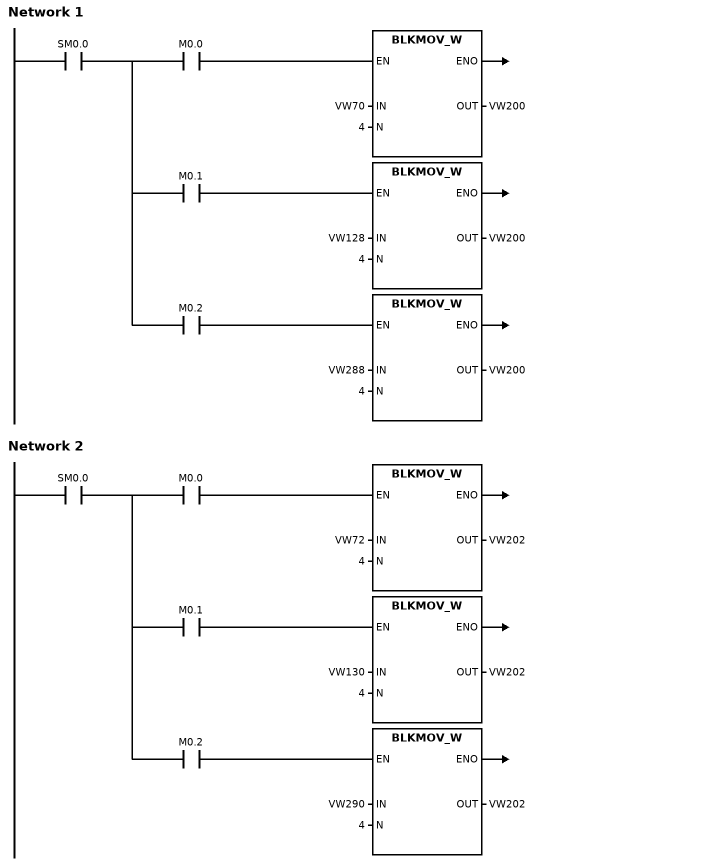
Network 1
LD     SM0.0
LPS
A      M0.0
BMW    VW70, VW200, 4
LRD
A      M0.1
BMW    VW128, VW200, 4
LPP
A      M0.2
BMW    VW288, VW200, 4
Network 2
LD     SM0.0
LPS
A      M0.0
BMW    VW72, VW202, 4
LRD
A      M0.1
BMW    VW130, VW202, 4
LPP
A      M0.2
BMW    VW290, VW202, 4
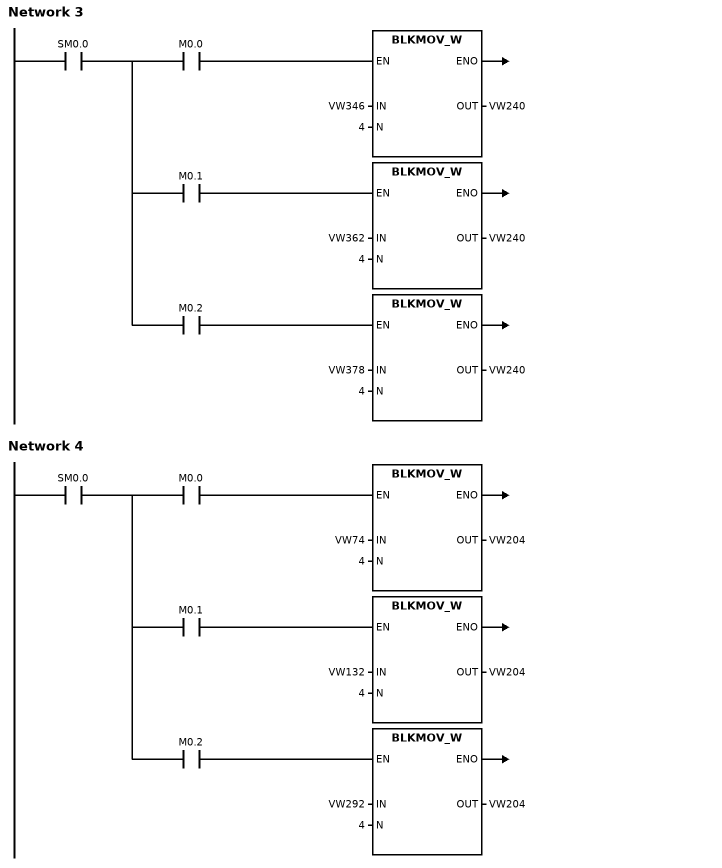
Network 3
LD     SM0.0
LPS
A      M0.0
BMW    VW346, VW240, 4
LRD
A      M0.1
BMW    VW362, VW240, 4
LPP
A      M0.2
BMW    VW378, VW240, 4
Network 4
LD     SM0.0
LPS
A      M0.0
BMW    VW74, VW204, 4
LRD
A      M0.1
BMW    VW132, VW204, 4
LPP
A      M0.2
BMW    VW292, VW204, 4
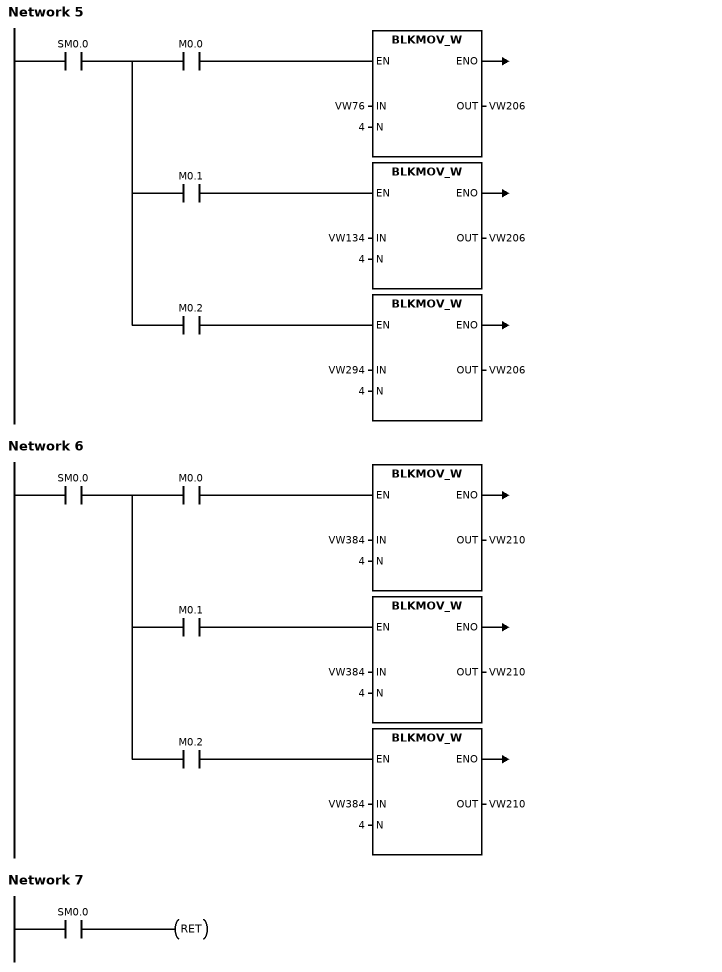
Network 5
LD     SM0.0
LPS
A      M0.0
BMW    VW76, VW206, 4
LRD
A      M0.1
BMW    VW134, VW206, 4
LPP
A      M0.2
BMW    VW294, VW206, 4
Network 6
LD     SM0.0
LPS
A      M0.0
BMW    VW384, VW210, 4
LRD
A      M0.1
BMW    VW384, VW210, 4
LPP
A      M0.2
BMW    VW384, VW210, 4
Network 7
LD     SM0.0
CRET
END_SUBROUTINE_BLOCK

SUBROUTINE_BLOCK thoidiem7:SBR9
TITLE=
BEGIN
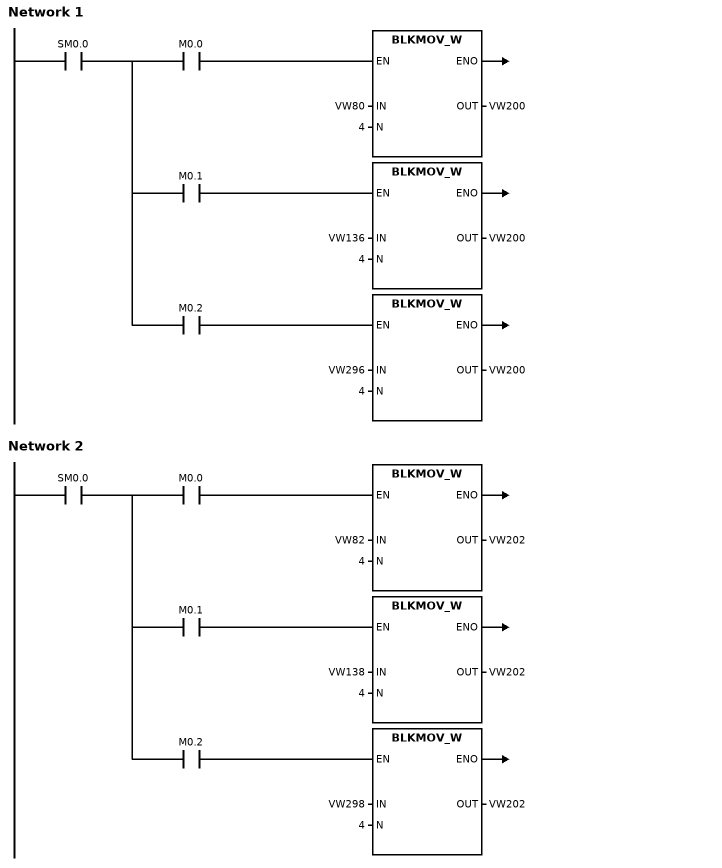
Network 1
LD     SM0.0
LPS
A      M0.0
BMW    VW80, VW200, 4
LRD
A      M0.1
BMW    VW136, VW200, 4
LPP
A      M0.2
BMW    VW296, VW200, 4
Network 2
LD     SM0.0
LPS
A      M0.0
BMW    VW82, VW202, 4
LRD
A      M0.1
BMW    VW138, VW202, 4
LPP
A      M0.2
BMW    VW298, VW202, 4
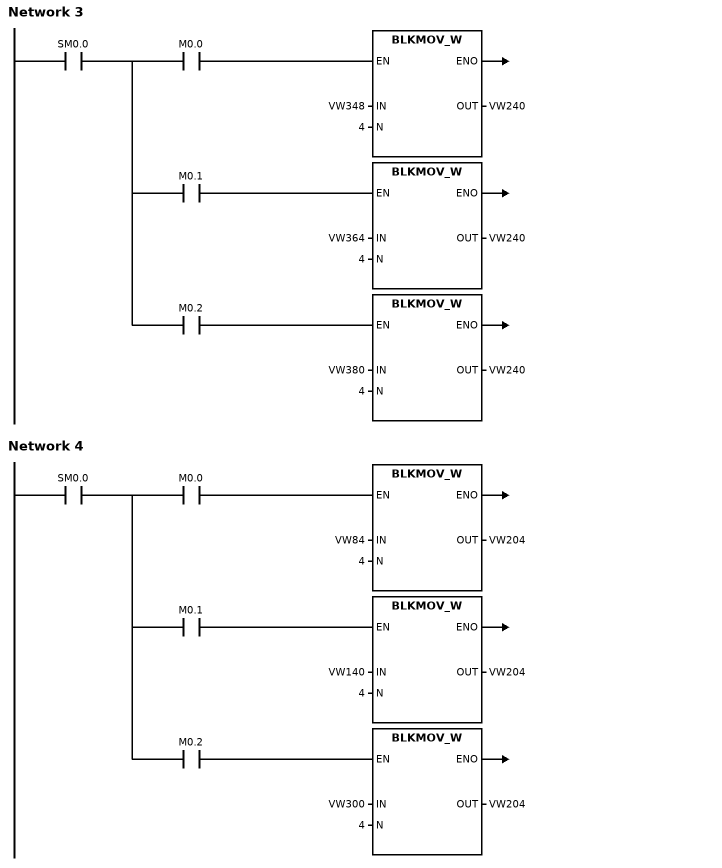
Network 3
LD     SM0.0
LPS
A      M0.0
BMW    VW348, VW240, 4
LRD
A      M0.1
BMW    VW364, VW240, 4
LPP
A      M0.2
BMW    VW380, VW240, 4
Network 4
LD     SM0.0
LPS
A      M0.0
BMW    VW84, VW204, 4
LRD
A      M0.1
BMW    VW140, VW204, 4
LPP
A      M0.2
BMW    VW300, VW204, 4
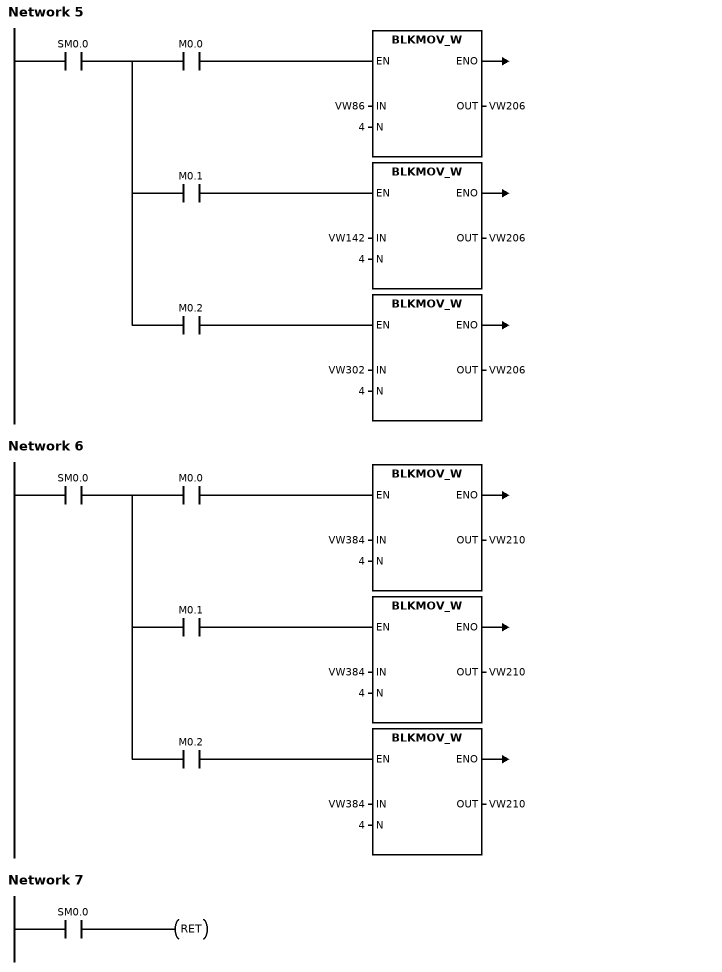
Network 5
LD     SM0.0
LPS
A      M0.0
BMW    VW86, VW206, 4
LRD
A      M0.1
BMW    VW142, VW206, 4
LPP
A      M0.2
BMW    VW302, VW206, 4
Network 6
LD     SM0.0
LPS
A      M0.0
BMW    VW384, VW210, 4
LRD
A      M0.1
BMW    VW384, VW210, 4
LPP
A      M0.2
BMW    VW384, VW210, 4
Network 7
LD     SM0.0
CRET
END_SUBROUTINE_BLOCK

SUBROUTINE_BLOCK tudong3phase:SBR10
TITLE=
BEGIN
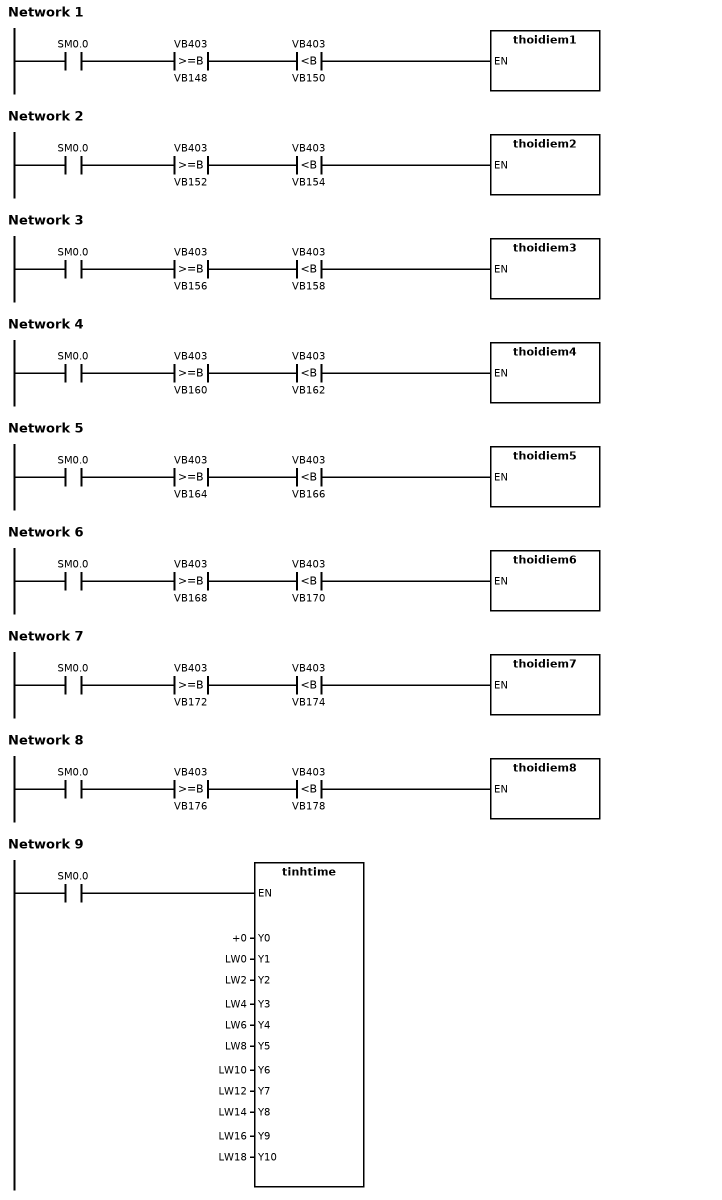
Network 1
LD     SM0.0
AB>=   VB403, VB148
AB<    VB403, VB150
CALL   thoidiem1:SBR3
Network 2
LD     SM0.0
AB>=   VB403, VB152
AB<    VB403, VB154
CALL   thoidiem2:SBR4
Network 3
LD     SM0.0
AB>=   VB403, VB156
AB<    VB403, VB158
CALL   thoidiem3:SBR5
Network 4
LD     SM0.0
AB>=   VB403, VB160
AB<    VB403, VB162
CALL   thoidiem4:SBR6
Network 5
LD     SM0.0
AB>=   VB403, VB164
AB<    VB403, VB166
CALL   thoidiem5:SBR7
Network 6
LD     SM0.0
AB>=   VB403, VB168
AB<    VB403, VB170
CALL   thoidiem6:SBR8
Network 7
LD     SM0.0
AB>=   VB403, VB172
AB<    VB403, VB174
CALL   thoidiem7:SBR9
Network 8
LD     SM0.0
AB>=   VB403, VB176
AB<    VB403, VB178
CALL   thoidiem8:SBR14
Network 9
LD     SM0.0
CALL   tinhtime:SBR16, +0, LW0, LW2, LW4, LW6, LW8, LW10, LW12, LW14, LW16, LW18
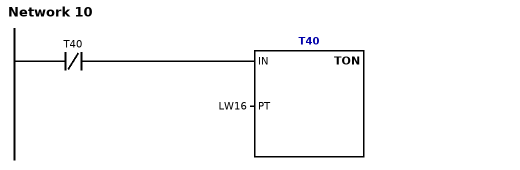
Network 10
LDN    T40
TON    T40, LW16
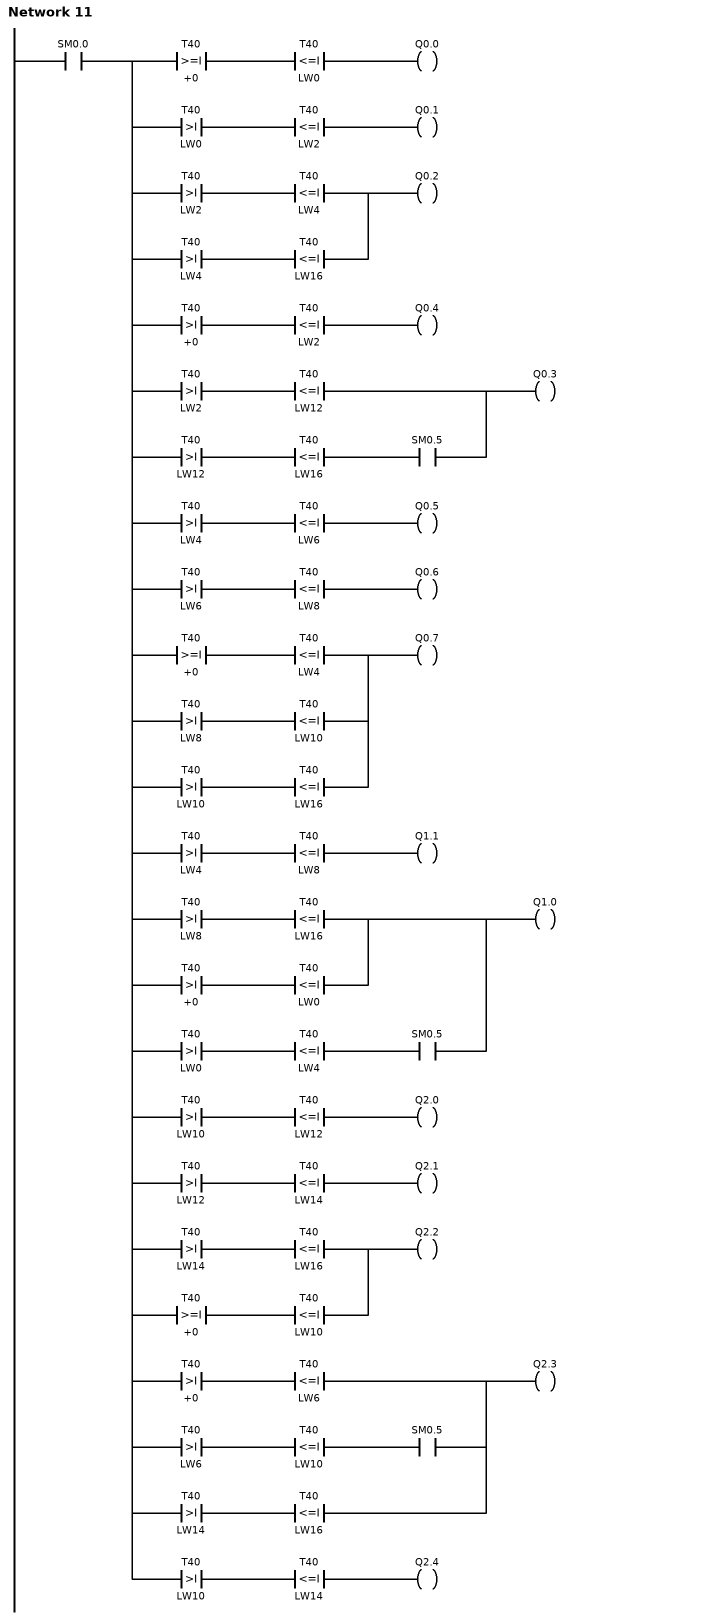
Network 11
LD     SM0.0
LPS
AW>=   T40, +0
AW<=   T40, LW0
=      Q0.0
LRD
AW>    T40, LW0
AW<=   T40, LW2
=      Q0.1
LRD
LDW>   T40, LW2
AW<=   T40, LW4
LDW>   T40, LW4
AW<=   T40, LW16
OLD
ALD
=      Q0.2
LRD
AW>    T40, +0
AW<=   T40, LW2
=      Q0.4
LRD
LDW>   T40, LW2
AW<=   T40, LW12
LDW>   T40, LW12
AW<=   T40, LW16
A      SM0.5
OLD
ALD
=      Q0.3
LRD
LPS
AW>    T40, LW4
AW<=   T40, LW6
=      Q0.5
LPP
AW>    T40, LW6
AW<=   T40, LW8
=      Q0.6
LRD
LDW>=  T40, +0
AW<=   T40, LW4
LDW>   T40, LW8
AW<=   T40, LW10
OLD
LDW>   T40, LW10
AW<=   T40, LW16
OLD
ALD
=      Q0.7
LRD
AW>    T40, LW4
AW<=   T40, LW8
=      Q1.1
LRD
LDW>   T40, LW8
AW<=   T40, LW16
LDW>   T40, +0
AW<=   T40, LW0
OLD
LDW>   T40, LW0
AW<=   T40, LW4
A      SM0.5
OLD
ALD
=      Q1.0
LRD
LPS
AW>    T40, LW10
AW<=   T40, LW12
=      Q2.0
LPP
AW>    T40, LW12
AW<=   T40, LW14
=      Q2.1
LRD
LDW>   T40, LW14
AW<=   T40, LW16
LDW>=  T40, +0
AW<=   T40, LW10
OLD
ALD
=      Q2.2
LRD
LDW>   T40, +0
AW<=   T40, LW6
LDW>   T40, LW6
AW<=   T40, LW10
A      SM0.5
OLD
LDW>   T40, LW14
AW<=   T40, LW16
OLD
ALD
=      Q2.3
LPP
AW>    T40, LW10
AW<=   T40, LW14
=      Q2.4
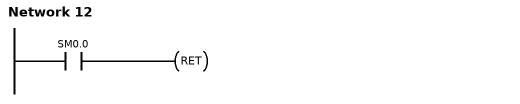
Network 12
LD     SM0.0
CRET
END_SUBROUTINE_BLOCK

SUBROUTINE_BLOCK chonngay:SBR11
TITLE=
BEGIN
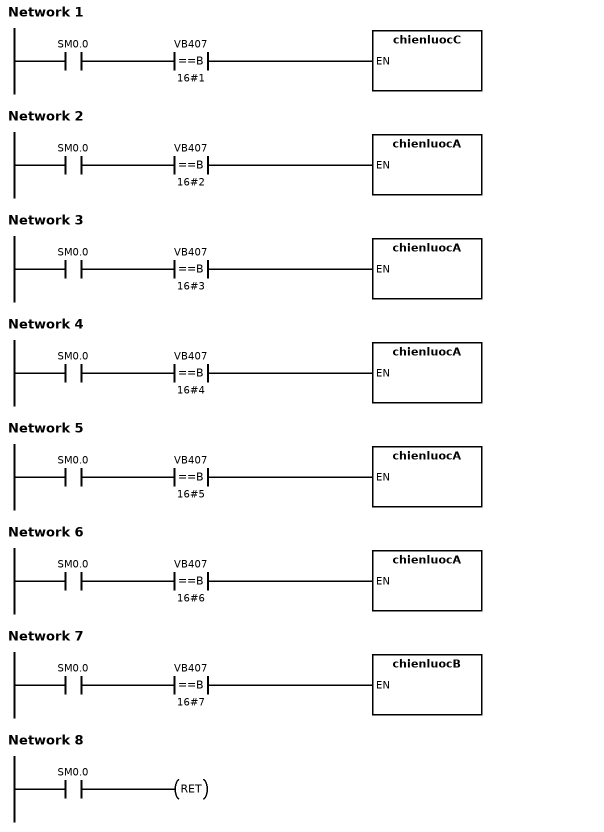
Network 1
LD     SM0.0
AB=    VB407, 16#1
CALL   chienluocC:SBR15
Network 2
LD     SM0.0
AB=    VB407, 16#2
CALL   chienluocA:SBR12
Network 3
LD     SM0.0
AB=    VB407, 16#3
CALL   chienluocA:SBR12
Network 4
LD     SM0.0
AB=    VB407, 16#4
CALL   chienluocA:SBR12
Network 5
LD     SM0.0
AB=    VB407, 16#5
CALL   chienluocA:SBR12
Network 6
LD     SM0.0
AB=    VB407, 16#6
CALL   chienluocA:SBR12
Network 7
LD     SM0.0
AB=    VB407, 16#7
CALL   chienluocB:SBR13
Network 8
LD     SM0.0
CRET
END_SUBROUTINE_BLOCK

SUBROUTINE_BLOCK chienluocA:SBR12
TITLE=
BEGIN
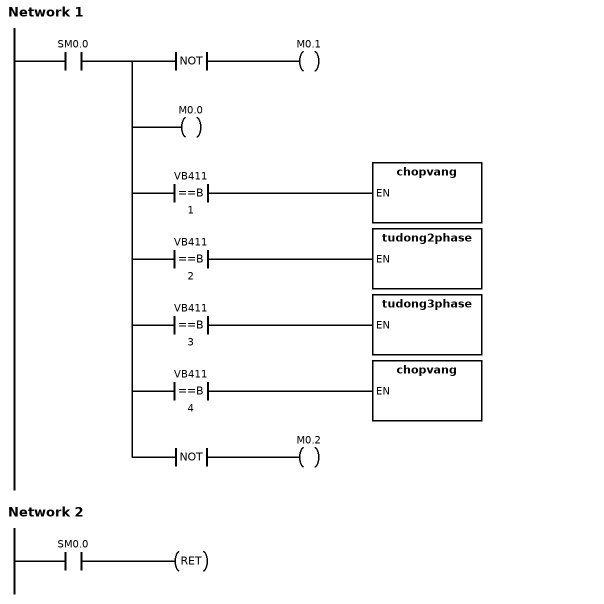
Network 1
LD     SM0.0
LPS
NOT
=      M0.1
LRD
=      M0.0
LRD
AB=    VB411, 1
CALL   chopvang:SBR1
LRD
AB=    VB411, 2
CALL   tudong2phase:SBR0
LRD
AB=    VB411, 3
CALL   tudong3phase:SBR10
LRD
AB=    VB411, 4
CALL   chopvang:SBR1
LPP
NOT
=      M0.2
Network 2
LD     SM0.0
CRET
END_SUBROUTINE_BLOCK

SUBROUTINE_BLOCK chienluocB:SBR13
TITLE=
BEGIN
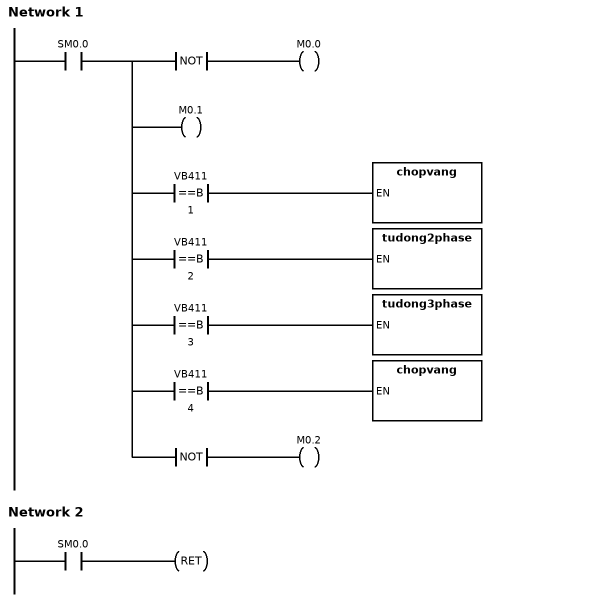
Network 1
LD     SM0.0
LPS
NOT
=      M0.0
LRD
=      M0.1
LRD
AB=    VB411, 1
CALL   chopvang:SBR1
LRD
AB=    VB411, 2
CALL   tudong2phase:SBR0
LRD
AB=    VB411, 3
CALL   tudong3phase:SBR10
LRD
AB=    VB411, 4
CALL   chopvang:SBR1
LPP
NOT
=      M0.2
Network 2
LD     SM0.0
CRET
END_SUBROUTINE_BLOCK

SUBROUTINE_BLOCK thoidiem8:SBR14
TITLE=
BEGIN
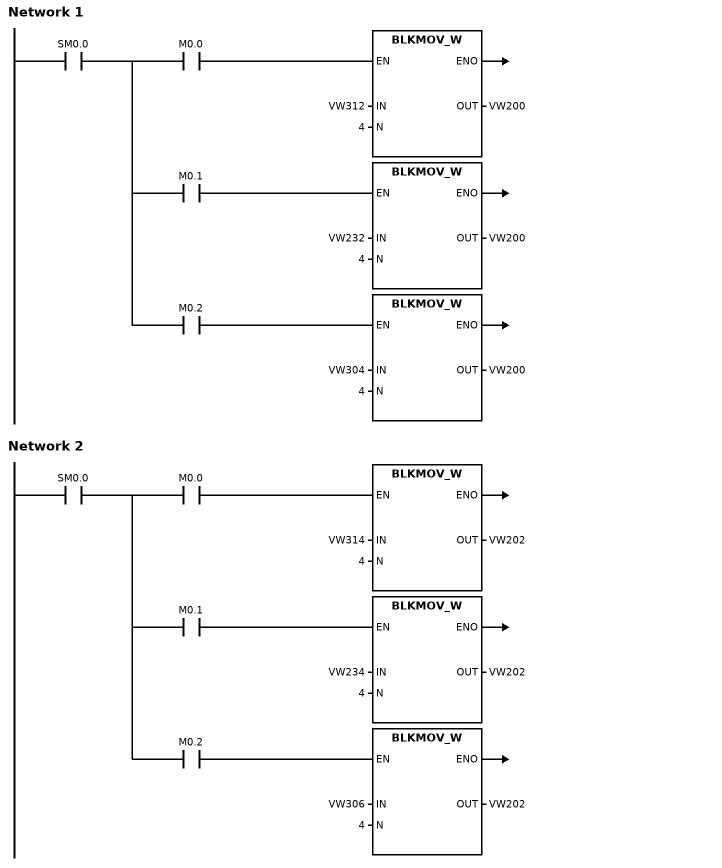
Network 1
LD     SM0.0
LPS
A      M0.0
BMW    VW312, VW200, 4
LRD
A      M0.1
BMW    VW232, VW200, 4
LPP
A      M0.2
BMW    VW304, VW200, 4
Network 2
LD     SM0.0
LPS
A      M0.0
BMW    VW314, VW202, 4
LRD
A      M0.1
BMW    VW234, VW202, 4
LPP
A      M0.2
BMW    VW306, VW202, 4
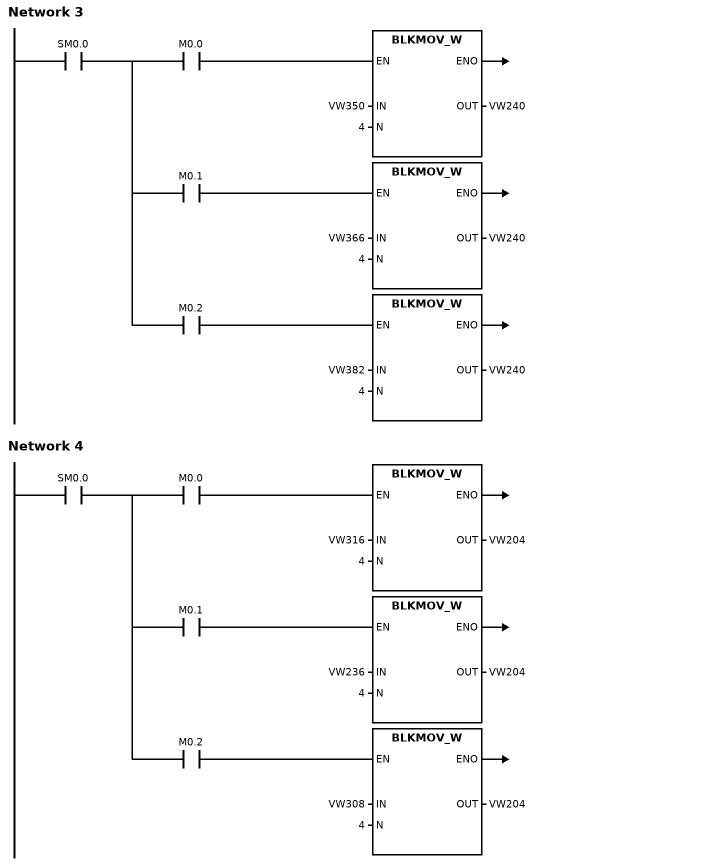
Network 3
LD     SM0.0
LPS
A      M0.0
BMW    VW350, VW240, 4
LRD
A      M0.1
BMW    VW366, VW240, 4
LPP
A      M0.2
BMW    VW382, VW240, 4
Network 4
LD     SM0.0
LPS
A      M0.0
BMW    VW316, VW204, 4
LRD
A      M0.1
BMW    VW236, VW204, 4
LPP
A      M0.2
BMW    VW308, VW204, 4
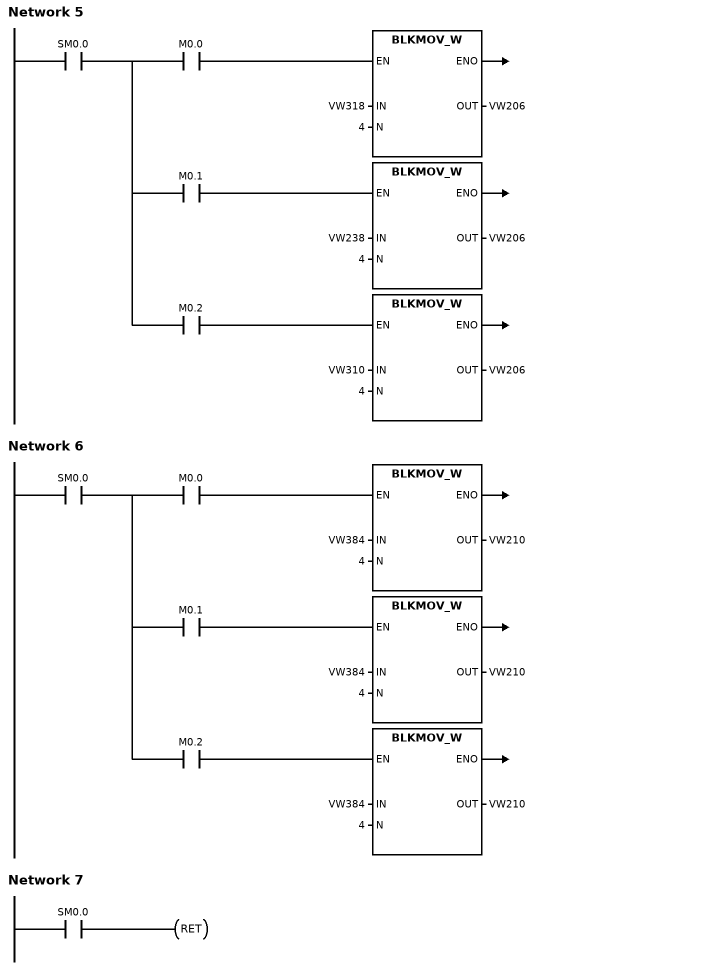
Network 5
LD     SM0.0
LPS
A      M0.0
BMW    VW318, VW206, 4
LRD
A      M0.1
BMW    VW238, VW206, 4
LPP
A      M0.2
BMW    VW310, VW206, 4
Network 6
LD     SM0.0
LPS
A      M0.0
BMW    VW384, VW210, 4
LRD
A      M0.1
BMW    VW384, VW210, 4
LPP
A      M0.2
BMW    VW384, VW210, 4
Network 7
LD     SM0.0
CRET
END_SUBROUTINE_BLOCK

SUBROUTINE_BLOCK chienluocC:SBR15
TITLE=
BEGIN
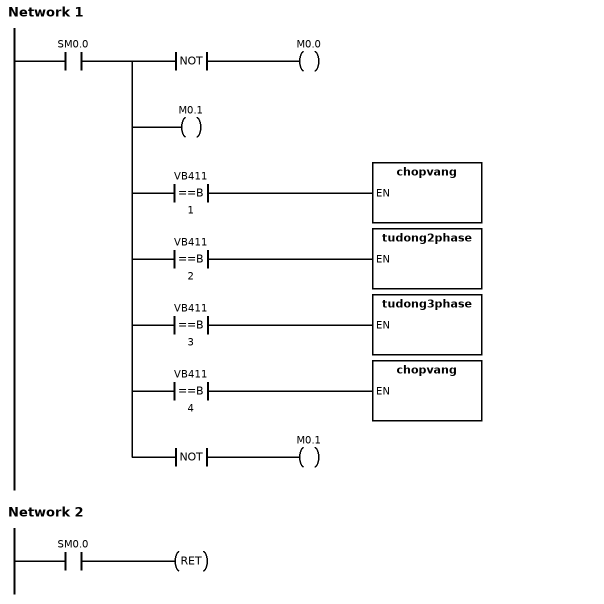
Network 1
LD     SM0.0
LPS
NOT
=      M0.0
LRD
=      M0.1
LRD
AB=    VB411, 1
CALL   chopvang:SBR1
LRD
AB=    VB411, 2
CALL   tudong2phase:SBR0
LRD
AB=    VB411, 3
CALL   tudong3phase:SBR10
LRD
AB=    VB411, 4
CALL   chopvang:SBR1
LPP
NOT
=      M0.1
Network 2
LD     SM0.0
CRET
END_SUBROUTINE_BLOCK

SUBROUTINE_BLOCK tinhtime:SBR16
TITLE=
VAR_INPUT
Y0:INT;	// LW0 
END_VAR
VAR_IN_OUT
Y1:INT;	// LW2 
Y2:INT;	// LW4 
Y3:INT;	// LW6 
Y4:INT;	// LW8 
Y5:INT;	// LW10 
Y6:INT;	// LW12 
Y7:INT;	// LW14 
Y8:INT;	// LW16 
Y9:INT;	// LW18 
Y10:INT;	// LW20 
END_VAR
BEGIN
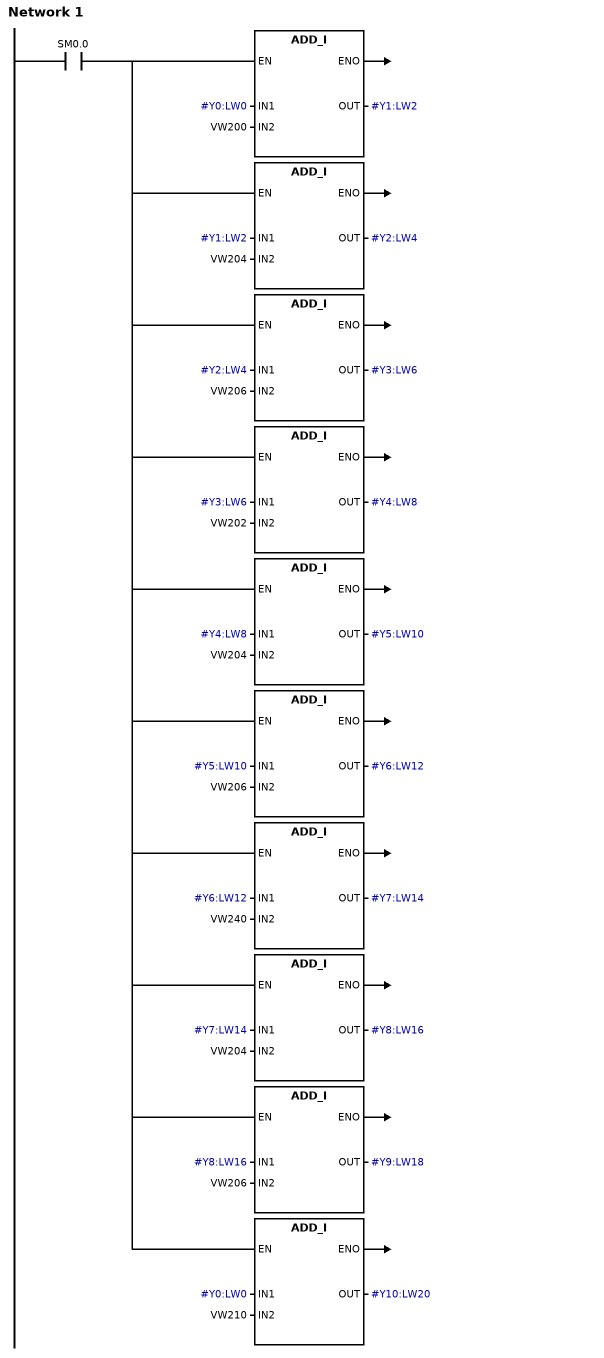
Network 1
LD     SM0.0
MOVW   #Y0:LW0, #Y1:LW2
+I     VW200, #Y1:LW2
MOVW   #Y1:LW2, #Y2:LW4
+I     VW204, #Y2:LW4
MOVW   #Y2:LW4, #Y3:LW6
+I     VW206, #Y3:LW6
MOVW   #Y3:LW6, #Y4:LW8
+I     VW202, #Y4:LW8
MOVW   #Y4:LW8, #Y5:LW10
+I     VW204, #Y5:LW10
MOVW   #Y5:LW10, #Y6:LW12
+I     VW206, #Y6:LW12
MOVW   #Y6:LW12, #Y7:LW14
+I     VW240, #Y7:LW14
MOVW   #Y7:LW14, #Y8:LW16
+I     VW204, #Y8:LW16
MOVW   #Y8:LW16, #Y9:LW18
+I     VW206, #Y9:LW18
MOVW   #Y0:LW0, #Y10:LW20
+I     VW210, #Y10:LW20
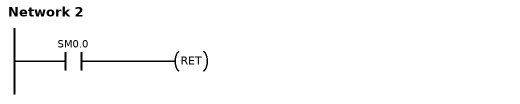
Network 2
LD     SM0.0
CRET
END_SUBROUTINE_BLOCK

DATA_BLOCK_TAB USER1
BEGIN
VW20     +250
VW22     +250
VW24     +30
VW26     +30
VW30     +250
VW32     +250
VW34     +30
VW36     +30
VW40     +250
VW42     +250
VW44     +30
VW46     +30
VW50     +250
VW52     +250
VW54     +30
VW56     +30
VW60     +250
VW62     +250
VW64     +30
VW66     +30
VW70     +250
VW72     +250
VW74     +30
VW76     +30
VW80     +250
VW82     +250
VW84     +30
VW86     +30
VW88     +250
VW90     +250
VW92     +30
VW94     +30
VW96     +250
VW98     +250
VW100    +30
VW102    +30
VW104    +250
VW106    +250
VW108    +30
VW110    +30
VW112    +250
VW114    +250
VW116    +30
VW118    +30
VW120    +250
VW122    +250
VW124    +30
VW126    +30
VW128    +250
VW130    +250
VW132    +30
VW134    +30
VW136    +250
VW138    +250
VW140    +30
VW142    +30
VB144    16#5
VB145    16#0
VB146    16#23
VB147    16#0
VB148    16#6
VB149    16#0
VB150    16#8
VB151    16#0
VB152    16#8
VB154    16#11
VB156    16#11
VB158    16#13
VB160    16#13
VB162    16#17
VB164    16#17
VB166    16#18
VB168    16#18
VB170    16#20
VB172    16#20
VB174    16#21
VB176    16#21
VB178    16#22
VW232    +250
VW234    +250
VW236    +30
VW238    +30
VW248    +250
VW250    +250
VW252    +30
VW254    +30
VW256    +250
VW258    +250
VW260    +30
VW262    +30
VW264    +250
VW266    +250
VW268    +30
VW270    +30
VW272    +250
VW274    +250
VW276    +30
VW278    +30
VW280    +250
VW282    +250
VW284    +30
VW286    +30
VW288    +250
VW290    +250
VW292    +30
VW294    +30
VW296    +250
VW298    +250
VW300    +30
VW302    +30
VW304    +250
VW306    +250
VW308    +30
VW310    +30
VW312    +250
VW314    +250
VW316    +30
VW318    +30
VW332    +100
VW336    +250
VW338    +250
VW340    +250
VW342    +250
VW344    +250
VW346    +250
VW348    +250
VW350    +250
VW352    +250
VW354    +250
VW356    +250
VW358    +250
VW360    +250
VW362    +250
VW364    +250
VW366    +250
VW368    +250
VW370    +250
VW372    +250
VW374    +250
VW376    +250
VW378    +250
VW380    +250
VW382    +250
VW384    +50
VB409    16#0
VB410    16#0
VB411    16#2
VB412    16#0
END_DATA_BLOCK_TAB
